// TIA Portal V20 export
DATA_BLOCK "Data_From_Safety"   // DB21
{ S7_Optimized_Access := 'TRUE' }
// stored: MemoryReserve 100
   VAR
      Safety_Active : Bool;
      Safety_SS1 : Bool;
      Safety_SS2 : Bool;
      SS1_R1_1 : Bool;
      SS1_R1_2 : Bool;
      SS1_R2_1 : Bool;
      SS1_R2_2 : Bool;
      SS2_R1_1 : Bool;
      SS2_R1_2 : Bool;
      SS2_R2_1 : Bool;
      SS2_R2_2 : Bool;
      Estops : Array[0..14] of Bool;
   END_VAR
BEGIN
END_DATA_BLOCK
